// TIA Portal V17 export
// export: Created 2025-08-05T09:36:01.9075287Z, ExportSetting WithDefaults, DisplayName Totally Integrated Automation Portal, DisplayVersion V17, DisplayName TIA Portal Openness, DisplayVersion V17, DisplayName TIA Portal Version Control Interface, DisplayVersion V17, DisplayName SINAMICS Startdrive Advanced, DisplayVersion V17, DisplayName SINAMICS Startdrive G130, G150, S120, S150, SINAMICS MV, S210, DisplayVersion V17, DisplayName SINAMICS Startdrive G110M, G120, G120C, G120D, G120P, G115D, DisplayVersion V17, DisplayName STEP 7 Professional, DisplayVersion V17, DisplayName STEP 7 Safety, DisplayVersion V17, DisplayName WinCC Advanced, DisplayVersion V17
TYPE "YLS_Inputs"
// stored: IsFailsafeCompliant false
   STRUCT
      Laser_Assigned : Bool;   // Laser_Assigned
      Laser_On : Bool;   // Laser_On
      System_Error : Bool;   // System_Error
      Guide_Laser_On : Bool;   // Guide_Laser_On
      Program_Active : Bool;   // Program_Active
      End_of_Program : Bool;   // End_of_Program
      Program_Interrupted : Bool;   // Program_Interrupted
      Analogue_Control_On : Bool;   // Analogue_Control_On
      System_Warning : Bool;   // System_Warning
      Laser_Ready : Bool;   // Laser_Ready
      Emission_On : Bool;   // Emission_On
      Synchronization_Output : Bool;   // Synchronization_Output
      Robot_Mode : Bool;   // Robot_Mode
      Power_Supply_Interlock : Bool;   // Power_Supply_Interlock
      Laser_Enabled : Bool;   // Laser_Enabled
      LaserNet_Control : Bool;   // LaserNet_Control
      Output_Power : Int;   // Output_Power
      Optical_Channel : Byte;   // Optical_Channel
      Program_Number : Byte;   // Program_Number
      Laser_Error : Bool;   // Laser_Error
      Laser_Warning : Bool;   // Laser_Warning
      Chiller_Error : Bool;   // Chiller_Error
      Chiller_Warning : Bool;   // Chiller_Warning
      Safety_Interlock_Open : Bool;   // Safety_Interlock_Open
      Channel_Error : Bool;   // Channel_Error
      Laser_Busy : Bool;   // Laser_Busy
      Slot_Error : Bool;   // Slot_Error
      Cabinet_Door_Open : Bool;   // Cabinet_Door_Open
      Reserved_Option_On : Bool;   // Reserved_Option_On
      Reduced_Output_Power : Bool;   // Reduced_Output_Power
      High_Back_Reflection : Bool;   // High_Back_Reflection
      Module_Without_Voltage_Supply : Bool;   // Module_Without_Voltage_Supply
      Piercing_Mode : Bool;   // Piercing_Mode
      Single_Module_Mode : Bool;   // Single_Module_Mode
      Reserved : Bool;   // Reserved
      Laser_Number : Byte;   // Laser_Number
      Reserved_1 : Byte;   // Reserved_1
      Modules_Selection : Int;   // Modules_Selection
      Core_Modules_Actual_Power : Int;   // Core_Modules_Actual_Power
      Ring_Modules_Actual_Power : Int;   // Ring_Modules_Actual_Power
   END_STRUCT;
END_TYPE
